(* PLC project Untitled1.project, CODESYS CODESYS V3.5 SP8 Patch 2 *)
(* stored: creationDateTime 2016-04-18T22:24:28.5417761, modificationDateTime 2016-04-18T22:24:16.4690856 *)

PROGRAM StateInExample
  VAR
    input AT %IX0.0 : BOOL;
    output AT %QX0.0 : BOOL;
  END_VAR

                  
									output := input;
									
                
END_PROGRAM

PROGRAM Ontarto
  VAR
    input1 AT %IX0.0 : BOOL;
    stop AT %MX0.0 : BOOL;
    output AT %QX0.0 : BOOL;
  END_VAR

                  
									output := input1 OR output;
									IF
									 stop THEN output := FALSE;
									END_IF;
									
                
END_PROGRAM

PROGRAM Motor_Proba
  VAR_INPUT
    START AT %MX0.1 : BOOL := FALSE;
    STOP AT %MX0.2 : BOOL := FALSE;
  END_VAR
  VAR
    MOTOR AT %MX1.0 : BOOL := FALSE;
    ERROR AT %MX2.0 : BOOL := FALSE;
  END_VAR
  VAR
    ERR_TIM : TON;
    EL_TIME : TIME;
  END_VAR
  VAR_OUTPUT
    ST_RED AT %QX3.0 : BOOL;
    ST_GREEN AT %QX3.1 : BOOL;
  END_VAR

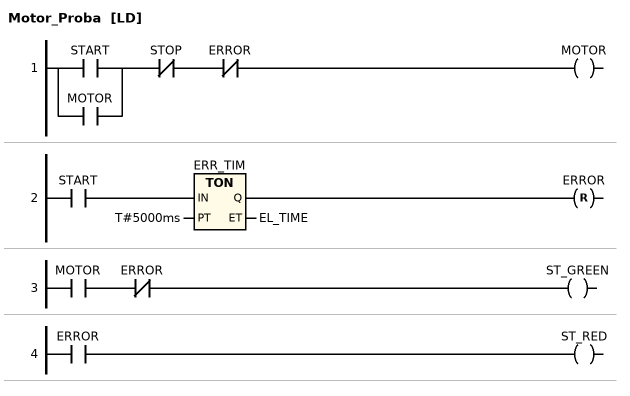
(* LD diagram, written out as Structured Text *)

MOTOR := (START OR MOTOR) AND NOT STOP AND NOT ERROR;

ERR_TIM(IN := START, PT := T#5000ms, ET => EL_TIME);
IF ERR_TIM.Q THEN ERROR := FALSE; END_IF;

ST_GREEN := MOTOR AND NOT ERROR;

ST_RED := ERROR;
END_PROGRAM

CONFIGURATION Application
  RESOURCE Application ON PLC
    TASK ExampleTask(INTERVAL := T#20ms, PRIORITY := 1);
    PROGRAM Motor_Proba WITH ExampleTask : Motor_Proba;
  END_RESOURCE
END_CONFIGURATION
